{attribute 'qualified_only'}
{attribute 'strict'}
TYPE E_PneumaticAxisGroup :
(
    ePneumaticAxisGroup1 := 1,
    ePneumaticAxisGroup2 := 2
) := ePneumaticAxisGroup1;
END_TYPE

(* stored: Version 1.1.0.1
   DUT E_PneumaticAxisGroup: Id {ddf4013f-9aa0-03e5-2424-e1247355bb7f} *)
